// TIA Portal V19 export
FUNCTION "Pb_Start_Presterilising" : Void   // FC60, STL
TITLE = Pb - PRESTERILIZING TANK
{ S7_Optimized_Access := 'TRUE' }
NAME : PBSTETNK
VERSION : 0.0
// Comment
// stored: AutoNumber false
   VAR_TEMP
      alarmbit : Int;
   END_VAR
BEGIN

NETWORK
TITLE = Pb - PRESTERILIZING TANK
      AN    "LEDAssignment".K3_BUTTON;  //"PbK3Presterilizing"
      BEC;
      R     "LEDAssignment".K3_BUTTON;  // "PbK3Presterilizing"
      A     "TANK AUTO";
      S     "ProcessAndPbAlarms"."A"[1];  //A01_TankInProcess// tank in process
      L     1;
      JC    Alrm;

//      BEC
      AN    "TANK CLEAN";
      S     "ProcessAndPbAlarms"."A"[2];  //A02_TankNotClean// not clean
      L     2;
      JC    Alrm;

//      BEC
      AN    "PA0572_Air";
      S     "ProcessAndPbAlarms"."A"[3];  //A03_NoInstrumentAir// no instument air
      L     3;
      JC    Alrm;

//      BEC
      AN    "PA0561_Steam";
      S     "ProcessAndPbAlarms"."A"[4];  //A04_NoSteam// no steam
      L     4;
      JC    Alrm;

//      BEC
      A     "DUMMY UPD.DRAIN TANK";
      S     "ProcessAndPbAlarms"."A"[5];  //A05_DrainIsActive// drain is active
      L     5;
      JC    Alrm;

//      BEC
      A(;
      AN    "GS22_61";
      A     "GS22_62";
      AN    "GS22_63";
      A     "GS22_68";
      O;
      A     "GS22_61";
      AN    "GS22_62";
      A     "GS22_63";
      AN    "GS22_68";
      );
      NOT;
      S     "ProcessAndPbAlarms"."A"[18];  //A18_SwingbendOutOfPosn// swingbend out of position
      L     6;
      JC    Alrm;

//      BEC
      S     "S0 PRESTERILIZING";
      S     "LEDAssignment".K3_LIGHT;  //"LIGHT_K3_PRESTE."
      R     "LEDAssignment".K3_FLASH;  //"FLASH_K3_PRESTE."
      BEU;

NETWORK
TITLE = Blockings alarm text
// Blockings alarm
Alrm: NOP   1;
      T     #alarmbit;
      CALL  "Set_Pop_Up_Blocking"
      ( alarmTextNum := #alarmbit
      );  // start blockings text


END_FUNCTION
